// TwinCAT 3 PLC project Hello_world
// ProgramVersion: 3.1.4026.18
// libraries:
//   Tc2_EtherCAT, * (Beckhoff Automation GmbH)
//   Tc2_Standard, * (Beckhoff Automation GmbH)
//   Tc2_System, * (Beckhoff Automation GmbH)
// project tree:
//   DUTs/ E_Command.TcDUT, E_PodState.TcDUT (not stored)
//   GVLs/ GVL_FSM.TcGVL (not stored), GVL_Levi.TcGVL, GVL_Prop.TcGVL (not stored), GVL_PT.TcGVL (not stored)
//   / PlcTask.TcTTO (not stored)
//   POUs/ BasicChecks.TcPOU (not stored), FB_Charge.TcPOU (not stored), CheckCritical.TcPOU (not stored), FB_Discharge.TcPOU (not stored), FB_Handle_Emergency.TcPOU, Handle_Movement.TcPOU (not stored), MAIN.TcPOU, Main_FSM.TcPOU (not stored)
// real-time tasks:
//   TASK PlcTask: cycle T#10ms, priority 20, ADS port 350
//   TASK HeartBeat: cycle T#10ms, priority 1, ADS port 351

// ---- DUTs/E_Command.TcDUT
{attribute 'qualified_only'}
{attribute 'strict'}
{attribute 'to_string'}
TYPE E_Command :
(
	CMD_NONE := 0,
    CMD_TO_IDLE,
    CMD_TO_HV_ACTIVE,
    CMD_TO_DEMO,
    CMD_TO_LEVITATION,
    CMD_TO_MOVEMENT,
    CMD_TO_MAINTENANCE,
    CMD_EMERGENCY
);
END_TYPE

// ---- GVLs/GVL_Levi.TcGVL
{attribute 'qualified_only'}
VAR_GLOBAL
	levitation_active:		BOOL;
	levitation_fault: 		BOOL;
	//DC link voltages
	drive_voltages: INT;
END_VAR

// ---- POUs/FB_Handle_Emergency.TcPOU
FUNCTION_BLOCK FB_Handle_Emergency
VAR_INPUT
    execute: 				BOOL;
END_VAR
VAR_OUTPUT
    busy: 					BOOL;
    done: 					BOOL;
END_VAR
VAR
    state: 					INT := 0;
    tonDelay: 				TON;
	allActionsComplete:		BOOL;
END_VAR

IF NOT execute THEN
    state := 0;
    busy := FALSE;
    done := FALSE;
    tonDelay(IN := FALSE);
    RETURN;
END_IF

//trigger EL!
busy := TRUE;
CASE state OF
    0:  GVL_FSM.open_SDC := TRUE;
        GVL_FSM.engage_brakes := TRUE;
        GVL_Prop.propulsion_enable := FALSE;
        GVL_Levi.levitation_active := FALSE;
        GVL_PT.emergency_shutdown := TRUE;
        state := 1;
        
    1:  allActionsComplete := 
            NOT GVL_FSM.sdc_closed AND
            GVL_FSM.brakes_engaged AND
            NOT GVL_Prop.propulsion_active AND
            NOT GVL_Levi.levitation_active;
        
        IF allActionsComplete THEN
            state := 2;
        END_IF
        
    2:	tonDelay(IN := TRUE, PT := T#200MS);
        IF tonDelay.Q THEN
            busy := FALSE;
            done := TRUE;
        END_IF
END_CASE

END_FUNCTION_BLOCK

// ---- POUs/MAIN.TcPOU
PROGRAM MAIN
VAR
	main_fsm	: Main_FSM;
END_VAR

main_fsm();

END_PROGRAM
